FUNCTION_BLOCK fb_LocalTime
VAR_INPUT

END_VAR
VAR_OUTPUT
  sLocalTime  : STRING;
  dtLocalTime : DT;
END_VAR
VAR
  GetSysTime    : FW_GetSystemTime;
  strFileTime   : T_FILETIME;
END_VAR

GetSysTime(dwTimeLo=> strFileTime.dwLowDateTime, dwTimeHi=> strFileTime.dwHighDateTime);

sLocalTime := SYSTEMTIME_TO_STRING( FILETIME_TO_SYSTEMTIME( strFileTime ) );
dtLocalTime := systemtime_to_dt( FILETIME_TO_SYSTEMTIME( strFileTime ) );

END_FUNCTION_BLOCK

(* stored: Version 1.1.0.1
   POU fb_LocalTime: Id {07812beb-d01a-4818-8dd7-3c3c8263a4bd}, SpecialFunc None *)
